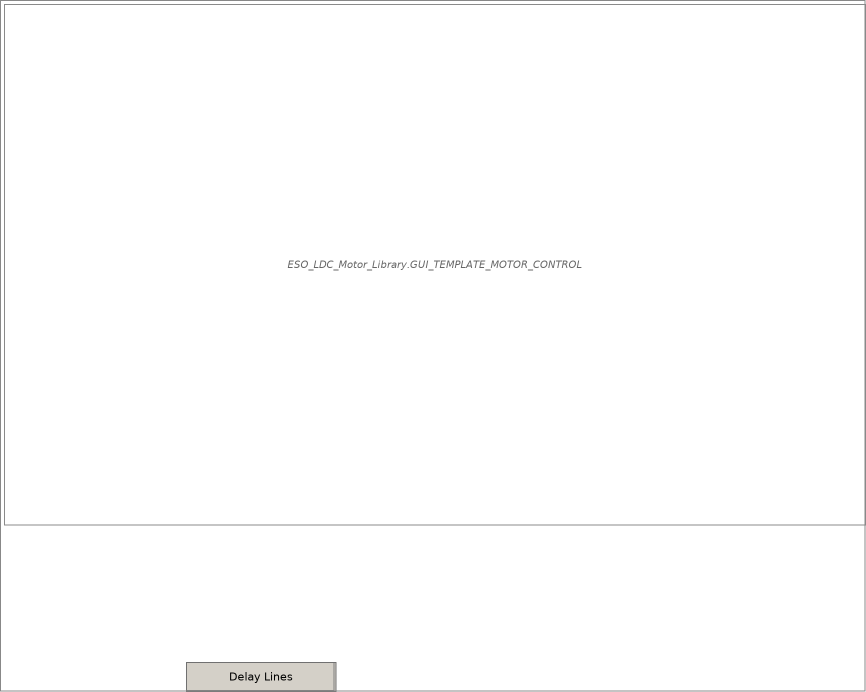
VISUALIZATION DL_MOTOR_01_CTRL  // 866x692
    Frame (4,4 862x521)
        shows ESO_LDC_Motor_Library.GUI_TEMPLATE_MOTOR_CONTROL(m_Instance := MAIN.DL_Motor_01)
    Button (186,662 150x30), "Delay Lines"
        OnMouseDown: change screen: SCIFY_Delay_Lines
END_VISUALIZATION

(* stored: Version 1.1.0.1, ProductVersion 3.1.4024.12
   Visu DL_MOTOR_01_CTRL: Id {32e912a3-e647-4356-b0dd-4edb717f74cb} *)
